// TIA Portal V20 export
// export: Created 2026-04-11T06:02:30.5682695Z, ExportSetting WithDefaults, DisplayName Totally Integrated Automation Portal, DisplayVersion V20, DisplayName TIA Portal Openness, DisplayVersion V20, DisplayName TIA Portal Version Control Interface, DisplayVersion V20, DisplayName STEP 7 Professional, DisplayVersion V20, DisplayName STEP 7 Safety, DisplayVersion V20, DisplayName WinCC Basic/Comfort/Advanced, DisplayVersion V20, DisplayName WinCC Unified, DisplayVersion V20
TYPE "udtHMI_MotorStarterET200"
// stored: IsFailsafeCompliant false
   STRUCT
      iMode : Int;
      iErrorCode { ExternalWritable := 'False'} : Int;
      iStatus { ExternalWritable := 'False'} : Int;
      rCurrent { ExternalWritable := 'False'} : Real;
      bPB_ResetError : Bool;
      bPB_Forward : Bool;
      bPB_Reverse : Bool;
      bPB_Stop : Bool;
      bPBEN_ResetError { ExternalWritable := 'False'} : Bool;
      bPBEN_Forward { ExternalWritable := 'False'} : Bool;
      bPBEN_Reverse { ExternalWritable := 'False'} : Bool;
      bPBEN_Stop { ExternalWritable := 'False'} : Bool;
      bForwardOn { ExternalWritable := 'False'} : Bool;
      bReverseOn { ExternalWritable := 'False'} : Bool;
      bSignalForward { ExternalWritable := 'False'} : Bool;
      bSignalReverse { ExternalWritable := 'False'} : Bool;
      bError { ExternalWritable := 'False'} : Bool;
      bInterlock { ExternalWritable := 'False'} : Bool;
      bInput1 { ExternalWritable := 'False'} : Bool;
      bInput2 { ExternalWritable := 'False'} : Bool;
      bInput3 { ExternalWritable := 'False'} : Bool;
      bManualLocalMode { ExternalWritable := 'False'} : Bool;
      bFailsafeStatus { ExternalWritable := 'False'} : Bool;
   END_STRUCT;
END_TYPE
